TYPE ST_Strings :
STRUCT
	(* Twelve strings used to store sample names *)
	{attribute 'pytmc' := '
        pv: 01
		io: i
     '}
	 s1 : STRING;
	 {attribute 'pytmc' := '
        pv: 02
		io: i
     '}
	 s2 : STRING;
	 {attribute 'pytmc' := '
        pv: 03
		io: i
     '}
	 s3 : STRING;
	 {attribute 'pytmc' := '
        pv: 04
		io: i
     '}
	 s4 : STRING;
	 {attribute 'pytmc' := '
        pv: 05
		io: i
     '}
	 s5 : STRING;
	 {attribute 'pytmc' := '
        pv: 06
		io: i
     '}
	 s6 : STRING;
	 {attribute 'pytmc' := '
        pv: 07
		io: i
     '}
	 s7 : STRING;
	 {attribute 'pytmc' := '
        pv: 08
		io: i
     '}
	 s8 : STRING;
	 {attribute 'pytmc' := '
        pv: 09
		io: i
     '}
	 s9 : STRING;
	 {attribute 'pytmc' := '
        pv: 10
		io: i
     '}
	 s10 : STRING;
	 {attribute 'pytmc' := '
        pv: 11
		io: i
     '}
	 s11 : STRING;
	 {attribute 'pytmc' := '
        pv: 12
		io: i
     '}
	 s12 : STRING;
END_STRUCT
END_TYPE

(* stored: Version 1.1.0.1, ProductVersion 3.1.4022.18
   DUT ST_Strings: Id {732f2c27-82d7-468b-9b70-d5e6f1796e6b} *)
